% RSLogix 500 project LVD190111.RSS, saved by version 11.00.00.00 %
PROJECT "LINCEBOT"    % processor: MicroLogix 1400 %

PROGRAM FILES
  LAD 2 "MAIN"  43 rungs  % Main Program Routine %
  LAD 4 "PACKAGER"  10 rungs  % normal %
  LAD 6 "TIMING"  11 rungs  % normal %
  LAD 8 "LOOP TIME"  6 rungs
  LAD 10 "AIR PRESUR"  5 rungs
  LAD 12 "ENABLES"  10 rungs
  LAD 14 "SPEED OUT"  12 rungs
  LAD 16 "TOTALCOUNT"  4 rungs
  LAD 18 "TESTTRIG1"  3 rungs
  LAD 20 "TESTTRIG5"  3 rungs
  LAD 22 "TESTTRIG6"  3 rungs
  LAD 24 "NOTUSED"  1 rungs
  LAD 26 "TEST TIME"  11 rungs
  LAD 70 "NOTUSED"  3 rungs  % normal %
  LAD 80 "HSC BOT"  5 rungs
  LAD 90 "HSC TOP"  6 rungs
  LAD 100 "1 MS STI"  27 rungs  % high speed %
  LAD 102 "SPEED BOT"  8 rungs  % high speed %
  LAD 103 "SPEED TOP"  8 rungs  % high speed %
  LAD 104 "P BOT"  9 rungs  % high speed %
  LAD 105 "P TOP"  8 rungs  % high speed %
  LAD 110 "SHIFT BOT"  9 rungs
  LAD 111 "SHIFT TOP"  13 rungs
  LAD 122 "OPTICBOT"  2 rungs
  LAD 124 "INS1RESULT"  6 rungs
  LAD 125 "INS 1 MOVE"  7 rungs
  LAD 126 "INS 1TIME"  36 rungs
  LAD 127 "INS1"  16 rungs
  LAD 128 "INS1PASS"  4 rungs
  LAD 129 "INS1ACQ"  8 rungs
  LAD 130 "INS1TRIG"  5 rungs
  LAD 131 "XFER"  2 rungs
  LAD 141 "OPTICTOP"  13 rungs
  LAD 149 "INS5RESULT"  6 rungs
  LAD 150 "INS 5 MOVE"  11 rungs
  LAD 151 "INS 6 MOVE"  11 rungs
  LAD 152 "INS5"  16 rungs
  LAD 153 "INS5PASS"  4 rungs
  LAD 154 "INS5ACQ"  8 rungs
  LAD 155 "INS5TRIG"  5 rungs
  LAD 159 "INS6RESULT"  6 rungs
  LAD 160 "INS 5 TIME"  42 rungs
  LAD 161 "INS 6 TIME"  42 rungs
  LAD 162 "INS6"  16 rungs
  LAD 163 "INS6PASS"  4 rungs
  LAD 164 "INS6ACQ"  8 rungs
  LAD 165 "INS6TRIG"  5 rungs
  LAD 170 "PASS BLOW"  10 rungs
  LAD 180 "RATE"  9 rungs

DATA FILES
  O0 OUTPUT  11 elements
  I1 INPUT  11 elements
  S2 STATUS  66 elements
  B3 BINARY  14 elements
  T4 TIMER  40 elements
  C5 COUNTER  1 elements
  R6 CONTROL  20 elements
  N7 INTEGER  200 elements
  F8 FLOAT  100 elements
  B9 TOP BS DAT  256 elements
  B10 OLD_COM  1 elements
  B11 BOT BS DAT  256 elements
  B12 HMI_BINARY  22 elements  % general use with hmi to avoid additional reads %
  L13  COUNTS  100 elements
  F14 HMI_FLOATS  100 elements
  N15 HMI_INTS  100 elements
  L16 HMI_LONGS  100 elements
  B17 SIDE DATA  128 elements
  B18 TOP DATA  128 elements
  L19 INS1TIME  10 elements
  L20 INS1POS  10 elements
  L21 INS5TIME  10 elements
  L22 INS5POS  10 elements
  L23 NEW READ  100 elements
  L24 NEW WRITE  100 elements
  L25 INS6TIME  10 elements
  L26 INS6POS  10 elements
  L42   52 elements
  B181 BLANK  128 elements  % used to wipe bs files %
  F182 TEST FLOAT  50 elements
  L183 TEST LONG  50 elements
  N184 TEST INTS  50 elements
  B185 TEST BITS  50 elements
  N186 HMI INTS  50 elements
  L187 HMI LONG  50 elements
  F188 HMI FLOAT  50 elements
  B189 HMI BITS  50 elements
  L190 COUNTS  50 elements
  B191 ERROR BITS  10 elements
  L192 SPD OFFSET  50 elements
  F193 SPD OFFSET  50 elements
  B194 BOT GOOD  128 elements
  B195 TOP GOOD  128 elements
  B196 CTRL BITS  50 elements
  N197 CTRL INTS  50 elements
  B198 TRK BITS  50 elements
  L199 TRK LONG  50 elements
  N200 TRK INTS  50 elements
  L201 INS LONG  50 elements
  B202 INS BITS  50 elements
  N203 INS INTS  50 elements
  L204 CTRL LONG  50 elements
  F205 CTRL FLTS  50 elements

LADDER 2 "MAIN"    % Main Program Routine %
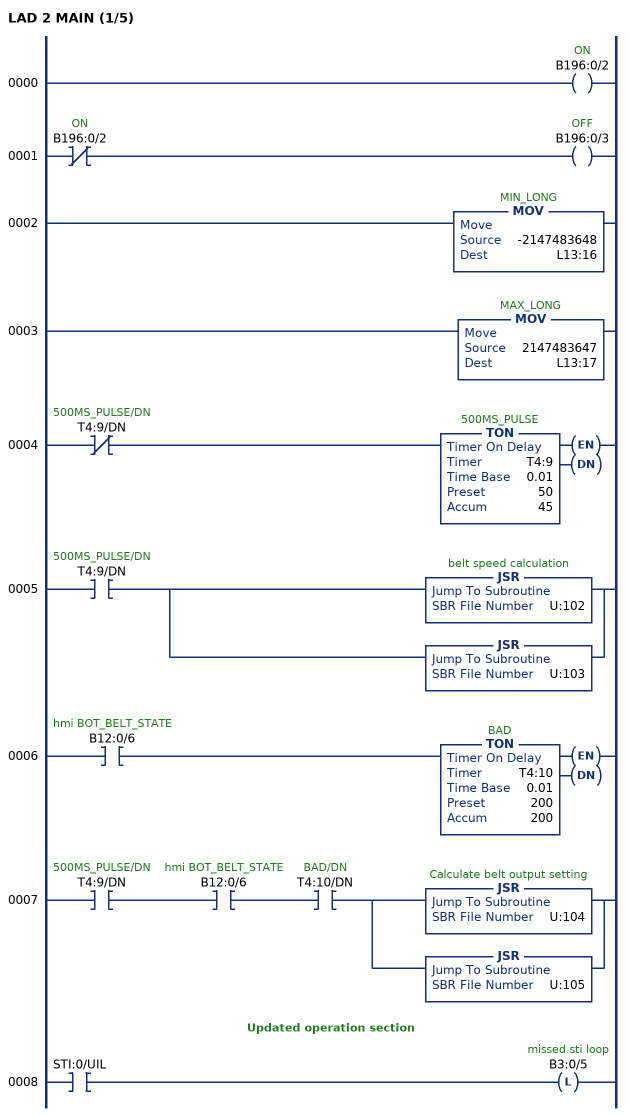
% Rung: 0 %
SOR OTE B196:0/2 EOR
%   B196:0/2  ON %
% Rung: 1 %
SOR XIO B196:0/2 OTE B196:0/3 EOR
%   B196:0/2  ON %
%   B196:0/3  OFF %
% Rung: 2 %
SOR MOV -2147483648 L13:16 EOR
%   L13:16  MIN_LONG %
% Rung: 3 %
SOR MOV 2147483647 L13:17 EOR
%   L13:17  MAX_LONG %
% Rung: 4 %
SOR XIO T4:9/DN TON T4:9 0.01 50 45 EOR
%   T4:9  500MS_PULSE %
% Rung: 5 %
SOR XIC T4:9/DN BST JSR U:102 NXB JSR U:103 BND EOR
%   T4:9  500MS_PULSE %
%   U:102  "belt speed calculation" %
% Rung: 6 %
SOR XIC B12:0/6 TON T4:10 0.01 200 200 EOR
%   B12:0/6  BOT_BELT_STATE  "hmi" %
%   T4:10  BAD %
% Rung: 7 %
SOR XIC T4:9/DN XIC B12:0/6 XIC T4:10/DN BST JSR U:104 NXB JSR U:105 BND EOR
%   T4:9  500MS_PULSE %
%   B12:0/6  BOT_BELT_STATE  "hmi" %
%   T4:10  BAD %
%   U:104  "Calculate belt output setting" %
% Rung: 8 %
% TITLE: Updated operation section %
SOR XIC STI:0/UIL OTL B3:0/5 EOR
%   B3:0/5  "missed sti loop" %

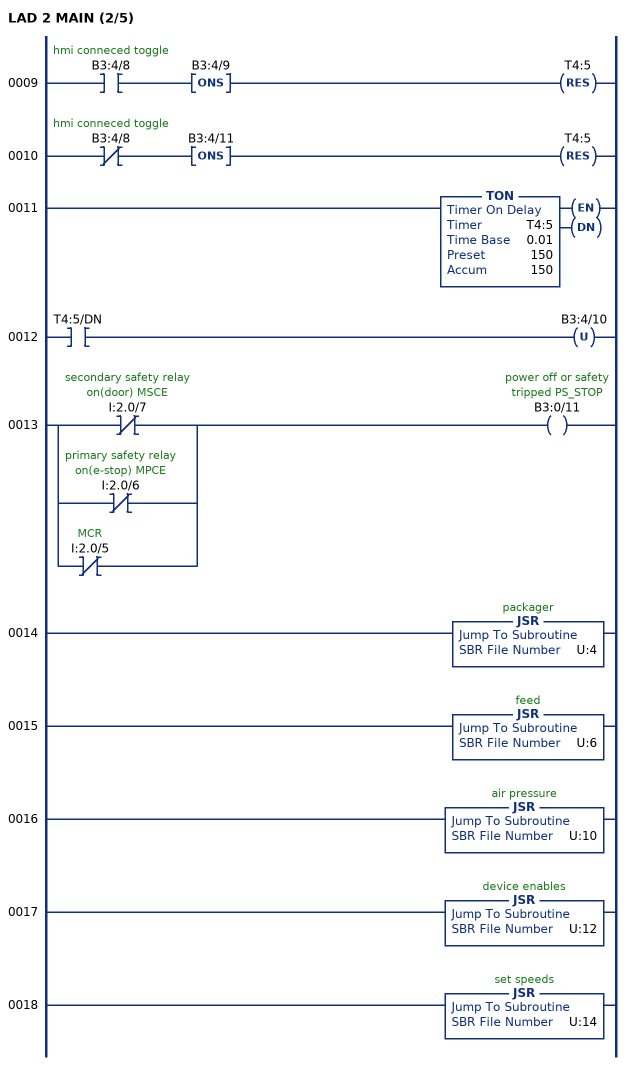
% Rung: 9 %
SOR XIC B3:4/8 ONS B3:4/9 RES T4:5 EOR
%   B3:4/8  "hmi conneced toggle" %
% Rung: 10 %
SOR XIO B3:4/8 ONS B3:4/11 RES T4:5 EOR
%   B3:4/8  "hmi conneced toggle" %
% Rung: 11 %
SOR TON T4:5 0.01 150 150 EOR
% Rung: 12 %
SOR XIC T4:5/DN OTU B3:4/10 EOR
% Rung: 13 %
SOR BST XIO I:2.0/7 NXB XIO I:2.0/6 NXB XIO I:2.0/5 BND OTE B3:0/11 EOR
%   I:2.0/7  MSCE  "secondary safety relay on(door)" %
%   I:2.0/6  MPCE  "primary safety relay on(e-stop)" %
%   I:2.0/5  MCR %
%   B3:0/11  PS_STOP  "power off or safety tripped" %
% Rung: 14 %
SOR JSR U:4 EOR
%   U:4  "packager" %
% Rung: 15 %
SOR JSR U:6 EOR
%   U:6  "feed" %
% Rung: 16 %
SOR JSR U:10 EOR
%   U:10  "air pressure" %
% Rung: 17 %
SOR JSR U:12 EOR
%   U:12  "device enables" %
% Rung: 18 %
SOR JSR U:14 EOR
%   U:14  "set speeds" %

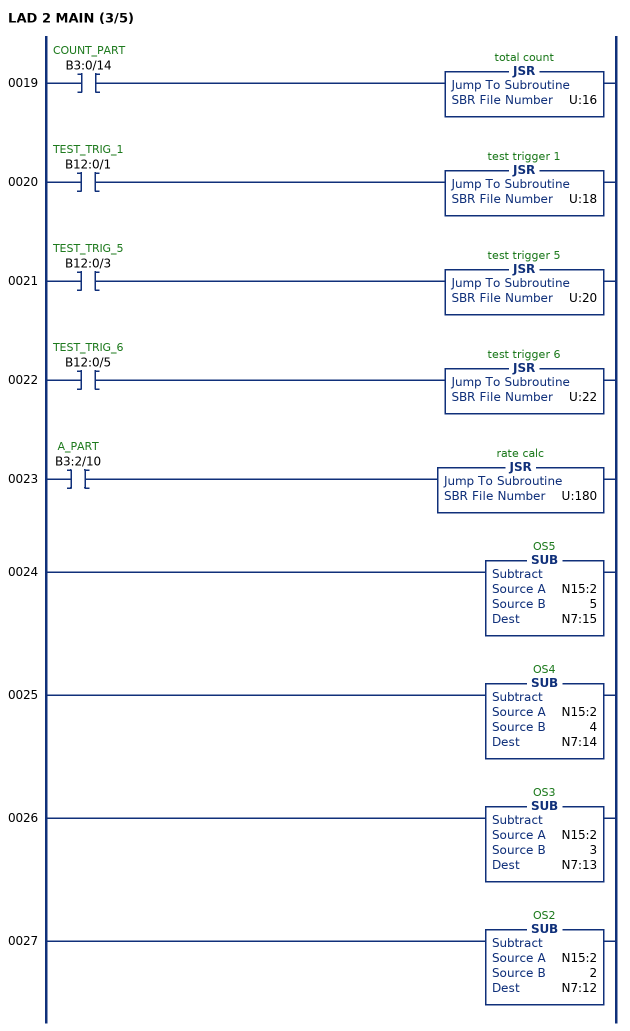
% Rung: 19 %
SOR XIC B3:0/14 JSR U:16 EOR
%   B3:0/14  COUNT_PART %
%   U:16  "total count" %
% Rung: 20 %
SOR XIC B12:0/1 JSR U:18 EOR
%   B12:0/1  TEST_TRIG_1 %
%   U:18  "test trigger 1" %
% Rung: 21 %
SOR XIC B12:0/3 JSR U:20 EOR
%   B12:0/3  TEST_TRIG_5 %
%   U:20  "test trigger 5" %
% Rung: 22 %
SOR XIC B12:0/5 JSR U:22 EOR
%   B12:0/5  TEST_TRIG_6 %
%   U:22  "test trigger 6" %
% Rung: 23 %
SOR XIC B3:2/10 JSR U:180 EOR
%   B3:2/10  A_PART %
%   U:180  "rate calc" %
% Rung: 24 %
SOR SUB N15:2 5 N7:15 EOR
%   N15:2  BLOW_PT %
%   N7:15  OS5 %
% Rung: 25 %
SOR SUB N15:2 4 N7:14 EOR
%   N15:2  BLOW_PT %
%   N7:14  OS4 %
% Rung: 26 %
SOR SUB N15:2 3 N7:13 EOR
%   N15:2  BLOW_PT %
%   N7:13  OS3 %
% Rung: 27 %
SOR SUB N15:2 2 N7:12 EOR
%   N15:2  BLOW_PT %
%   N7:12  OS2 %

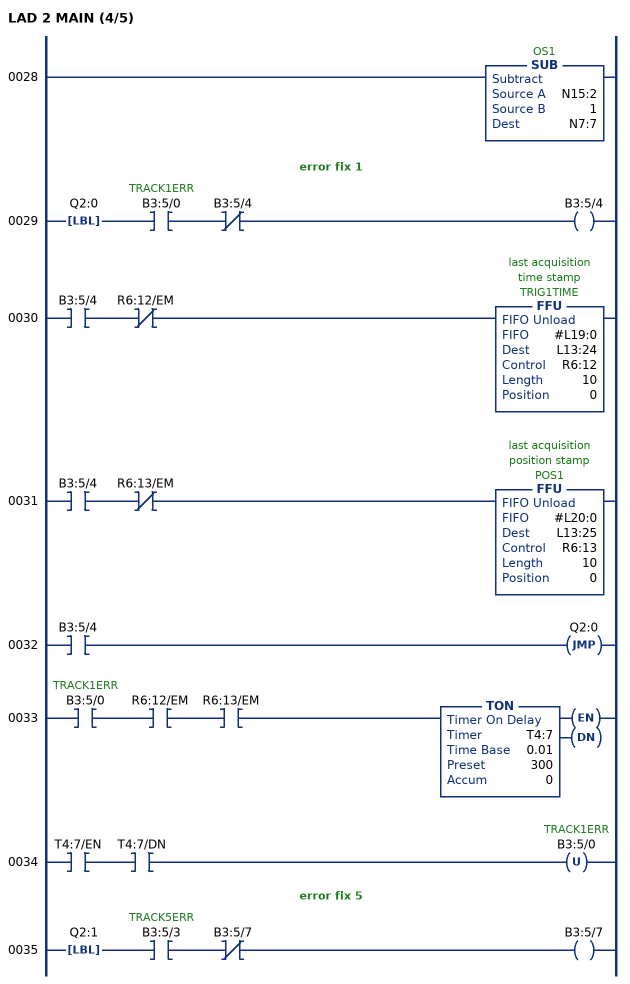
% Rung: 28 %
SOR SUB N15:2 1 N7:7 EOR
%   N15:2  BLOW_PT %
%   N7:7  OS1 %
% Rung: 29 %
% TITLE: error fix 1 %
SOR LBL Q2:0 XIC B3:5/0 XIO B3:5/4 OTE B3:5/4 EOR
%   B3:5/0  TRACK1ERR %
% Rung: 30 %
SOR XIC B3:5/4 XIO R6:12/EM FFU #L19:0 L13:24 R6:12 10 0 EOR
%   L13:24  TRIG1TIME  "last acquisition time stamp" %
% Rung: 31 %
SOR XIC B3:5/4 XIO R6:13/EM FFU #L20:0 L13:25 R6:13 10 0 EOR
%   L13:25  POS1  "last acquisition position stamp" %
% Rung: 32 %
SOR XIC B3:5/4 JMP Q2:0 EOR
% Rung: 33 %
SOR XIC B3:5/0 XIC R6:12/EM XIC R6:13/EM TON T4:7 0.01 300 0 EOR
%   B3:5/0  TRACK1ERR %
% Rung: 34 %
SOR XIC T4:7/EN XIC T4:7/DN OTU B3:5/0 EOR
%   B3:5/0  TRACK1ERR %
% Rung: 35 %
% TITLE: error fix 5 %
SOR LBL Q2:1 XIC B3:5/3 XIO B3:5/7 OTE B3:5/7 EOR
%   B3:5/3  TRACK5ERR %

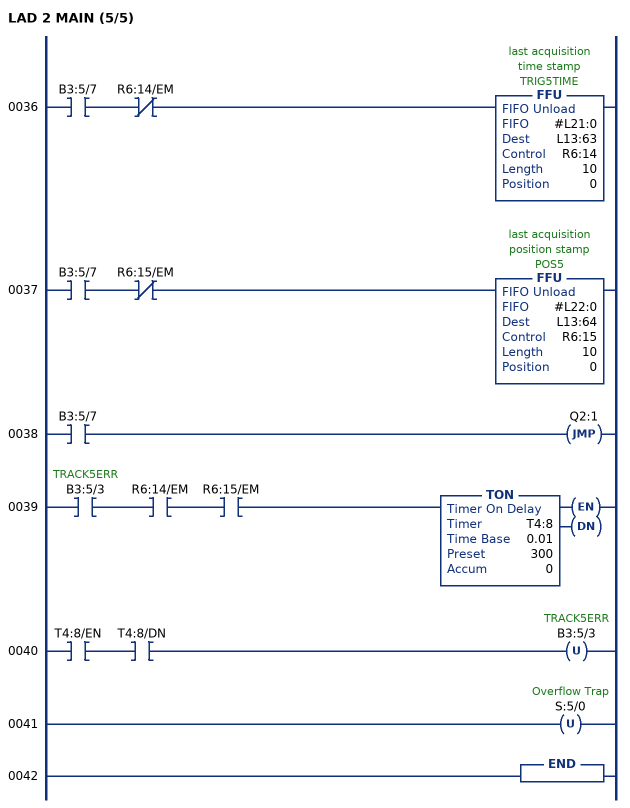
% Rung: 36 %
SOR XIC B3:5/7 XIO R6:14/EM FFU #L21:0 L13:63 R6:14 10 0 EOR
%   L13:63  TRIG5TIME  "last acquisition time stamp" %
% Rung: 37 %
SOR XIC B3:5/7 XIO R6:15/EM FFU #L22:0 L13:64 R6:15 10 0 EOR
%   L13:64  POS5  "last acquisition position stamp" %
% Rung: 38 %
SOR XIC B3:5/7 JMP Q2:1 EOR
% Rung: 39 %
SOR XIC B3:5/3 XIC R6:14/EM XIC R6:15/EM TON T4:8 0.01 300 0 EOR
%   B3:5/3  TRACK5ERR %
% Rung: 40 %
SOR XIC T4:8/EN XIC T4:8/DN OTU B3:5/3 EOR
%   B3:5/3  TRACK5ERR %
% Rung: 41 %
SOR OTU S:5/0 EOR
%   S:5/0  "Overflow Trap" %
% Rung: 42 %
SOR END EOR

LADDER 4 "PACKAGER"    % normal %
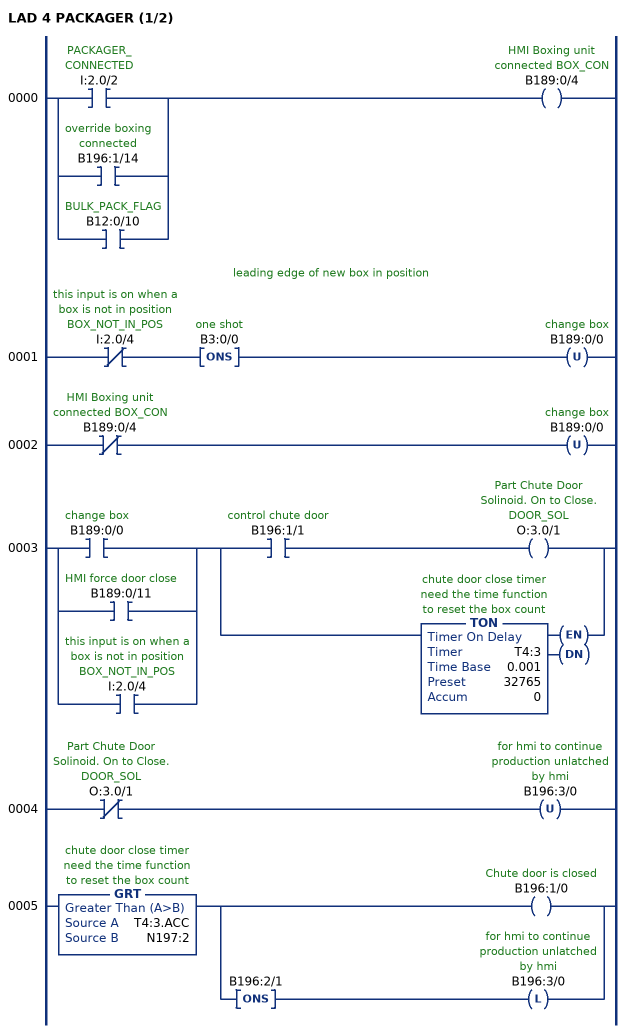
% Rung: 0 %
SOR BST XIC I:2.0/2 NXB XIC B196:1/14 NXB XIC B12:0/10 BND OTE B189:0/4 EOR
%   I:2.0/2  PACKAGER_CONNECTED %
%   B196:1/14  "override boxing connected" %
%   B12:0/10  BULK_PACK_FLAG %
%   B189:0/4  BOX_CON  "HMI Boxing unit connected" %
% Rung: 1 %
% leading edge of new box in position %
SOR XIO I:2.0/4 ONS B3:0/0 OTU B189:0/0 EOR
%   I:2.0/4  BOX_NOT_IN_POS  "this input is on when a box is not in position" %
%   B3:0/0  "one shot" %
%   B189:0/0  "change box" %
% Rung: 2 %
SOR XIO B189:0/4 OTU B189:0/0 EOR
%   B189:0/4  BOX_CON  "HMI Boxing unit connected" %
%   B189:0/0  "change box" %
% Rung: 3 %
SOR BST XIC B189:0/0 NXB XIC B189:0/11 NXB XIC I:2.0/4 BND BST XIC B196:1/1 OTE O:3.0/1 NXB TON T4:3 0.001 32765 0 BND EOR
%   B189:0/0  "change box" %
%   B189:0/11  "HMI force door close" %
%   I:2.0/4  BOX_NOT_IN_POS  "this input is on when a box is not in position" %
%   B196:1/1  "control chute door" %
%   O:3.0/1  DOOR_SOL  "Part Chute Door Solinoid. On to Close." %
%   T4:3  "chute door close timer need the time function to reset the box count" %
% Rung: 4 %
SOR XIO O:3.0/1 OTU B196:3/0 EOR
%   O:3.0/1  DOOR_SOL  "Part Chute Door Solinoid. On to Close." %
%   B196:3/0  "for hmi to continue production unlatched by hmi" %
% Rung: 5 %
SOR GRT T4:3.ACC N197:2 BST OTE B196:1/0 NXB ONS B196:2/1 OTL B196:3/0 BND EOR
%   T4:3  "chute door close timer need the time function to reset the box count" %
%   N197:2  "time for chute door to close" %
%   B196:1/0  "Chute door is closed" %
%   B196:3/0  "for hmi to continue production unlatched by hmi" %

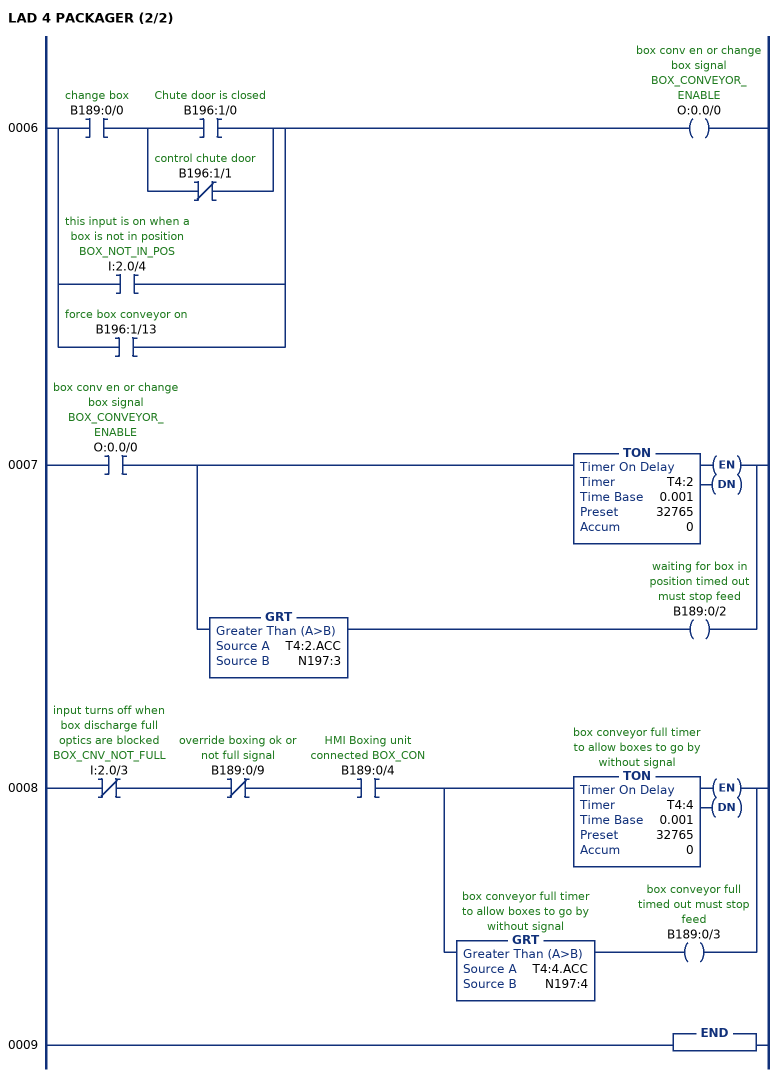
% Rung: 6 %
SOR BST XIC B189:0/0 BST XIC B196:1/0 NXB XIO B196:1/1 BND NXB XIC I:2.0/4 NXB XIC B196:1/13 BND OTE O:0.0/0 EOR
%   B189:0/0  "change box" %
%   B196:1/0  "Chute door is closed" %
%   B196:1/1  "control chute door" %
%   I:2.0/4  BOX_NOT_IN_POS  "this input is on when a box is not in position" %
%   B196:1/13  "force box conveyor on" %
%   O:0.0/0  BOX_CONVEYOR_ENABLE  "box conv en or change box signal" %
% Rung: 7 %
SOR XIC O:0.0/0 BST TON T4:2 0.001 32765 0 NXB GRT T4:2.ACC N197:3 OTE B189:0/2 BND EOR
%   O:0.0/0  BOX_CONVEYOR_ENABLE  "box conv en or change box signal" %
%   N197:3  "FeedWheel Speed Output Setting" %
%   B189:0/2  "waiting for box in position timed out must stop feed" %
% Rung: 8 %
SOR XIO I:2.0/3 XIO B189:0/9 XIC B189:0/4 BST TON T4:4 0.001 32765 0 NXB GRT T4:4.ACC N197:4 OTE B189:0/3 BND EOR
%   I:2.0/3  BOX_CNV_NOT_FULL  "input turns off when box discharge full optics are blocked" %
%   B189:0/9  "override boxing ok or not full signal" %
%   B189:0/4  BOX_CON  "HMI Boxing unit connected" %
%   T4:4  "box conveyor full timer to allow boxes to go by without signal" %
%   N197:4  "boxing convery full time out time (ms)" %
%   B189:0/3  "box conveyor full timed out must stop feed" %
% Rung: 9 %
SOR END EOR

LADDER 6 "TIMING"    % normal %
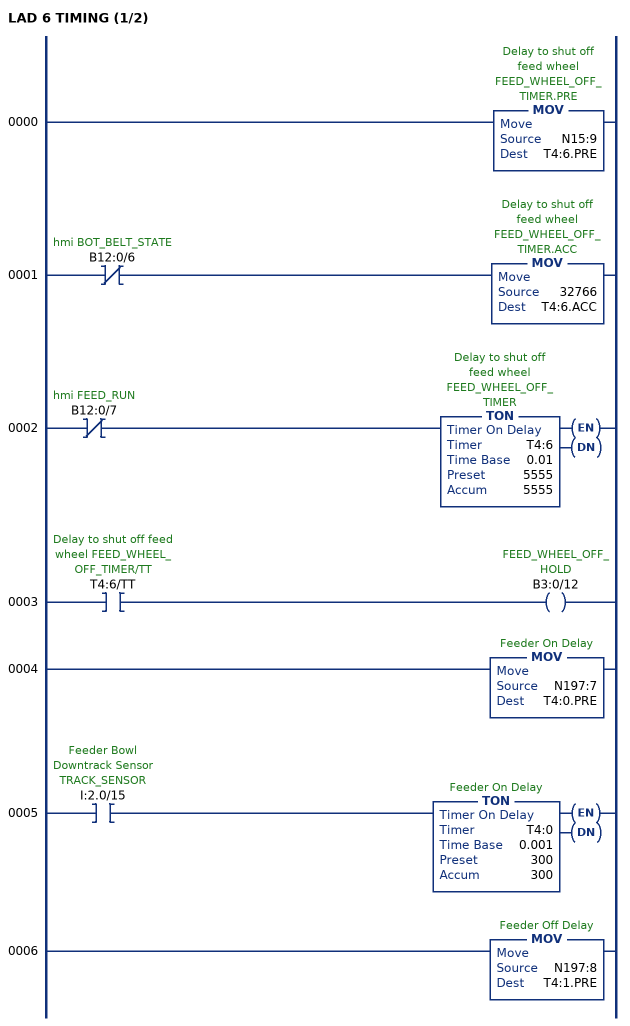
% Rung: 0 %
SOR MOV N15:9 T4:6.PRE EOR
%   N15:9  FEED_WHEEL_STOP_TIME %
%   T4:6  FEED_WHEEL_OFF_TIMER  "Delay to shut off feed wheel" %
% Rung: 1 %
SOR XIO B12:0/6 MOV 32766 T4:6.ACC EOR
%   B12:0/6  BOT_BELT_STATE  "hmi" %
%   T4:6  FEED_WHEEL_OFF_TIMER  "Delay to shut off feed wheel" %
% Rung: 2 %
SOR XIO B12:0/7 TON T4:6 0.01 5555 5555 EOR
%   B12:0/7  FEED_RUN  "hmi" %
%   T4:6  FEED_WHEEL_OFF_TIMER  "Delay to shut off feed wheel" %
% Rung: 3 %
SOR XIC T4:6/TT OTE B3:0/12 EOR
%   T4:6  FEED_WHEEL_OFF_TIMER  "Delay to shut off feed wheel" %
%   B3:0/12  FEED_WHEEL_OFF_HOLD %
% Rung: 4 %
SOR MOV N197:7 T4:0.PRE EOR
%   N197:7  "down track on delay" %
%   T4:0  "Feeder On Delay" %
% Rung: 5 %
SOR XIC I:2.0/15 TON T4:0 0.001 300 300 EOR
%   I:2.0/15  TRACK_SENSOR  "Feeder Bowl Downtrack Sensor" %
%   T4:0  "Feeder On Delay" %
% Rung: 6 %
SOR MOV N197:8 T4:1.PRE EOR
%   N197:8  "down track off delay" %
%   T4:1  "Feeder Off Delay" %

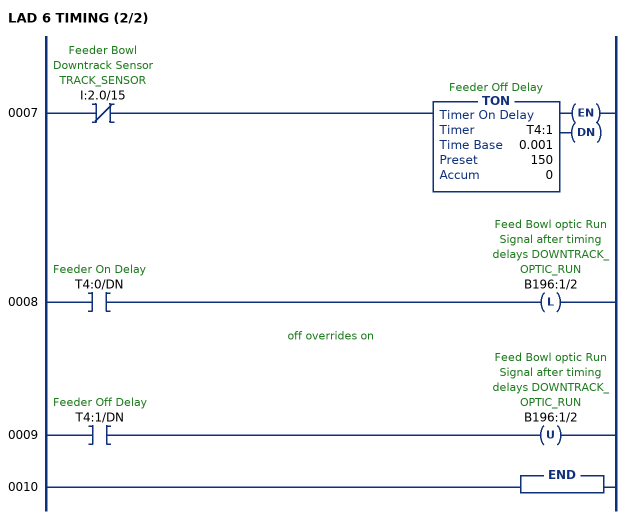
% Rung: 7 %
SOR XIO I:2.0/15 TON T4:1 0.001 150 0 EOR
%   I:2.0/15  TRACK_SENSOR  "Feeder Bowl Downtrack Sensor" %
%   T4:1  "Feeder Off Delay" %
% Rung: 8 %
SOR XIC T4:0/DN OTL B196:1/2 EOR
%   T4:0  "Feeder On Delay" %
%   B196:1/2  DOWNTRACK_OPTIC_RUN  "Feed Bowl optic Run Signal after timing delays" %
% Rung: 9 %
% off overrides on %
SOR XIC T4:1/DN OTU B196:1/2 EOR
%   T4:1  "Feeder Off Delay" %
%   B196:1/2  DOWNTRACK_OPTIC_RUN  "Feed Bowl optic Run Signal after timing delays" %
% Rung: 10 %
SOR END EOR

LADDER 8 "LOOP TIME"
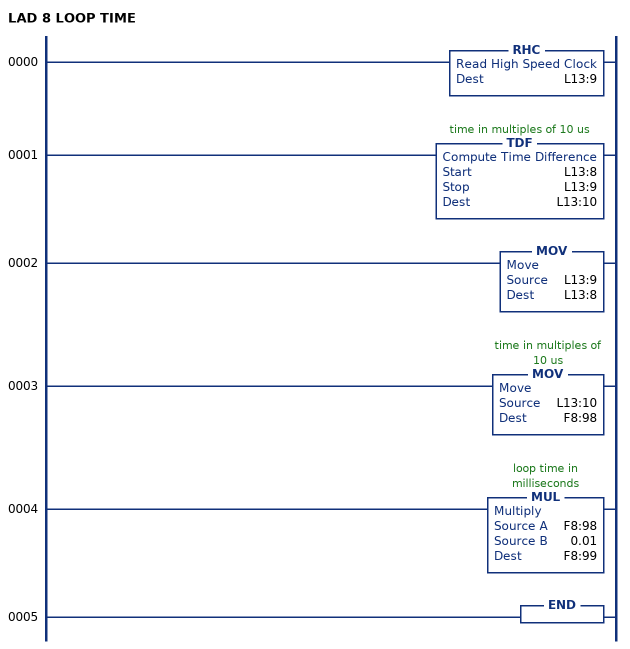
% Rung: 0 %
SOR RHC L13:9 EOR
% Rung: 1 %
SOR TDF L13:8 L13:9 L13:10 EOR
%   L13:10  "time in multiples of 10 us" %
% Rung: 2 %
SOR MOV L13:9 L13:8 EOR
% Rung: 3 %
SOR MOV L13:10 F8:98 EOR
%   L13:10  "time in multiples of 10 us" %
%   F8:98  "time in multiples of 10 us" %
% Rung: 4 %
SOR MUL F8:98 0.01 F8:99 EOR
%   F8:98  "time in multiples of 10 us" %
%   F8:99  "loop time in milliseconds" %
% Rung: 5 %
SOR END EOR

LADDER 10 "AIR PRESUR"
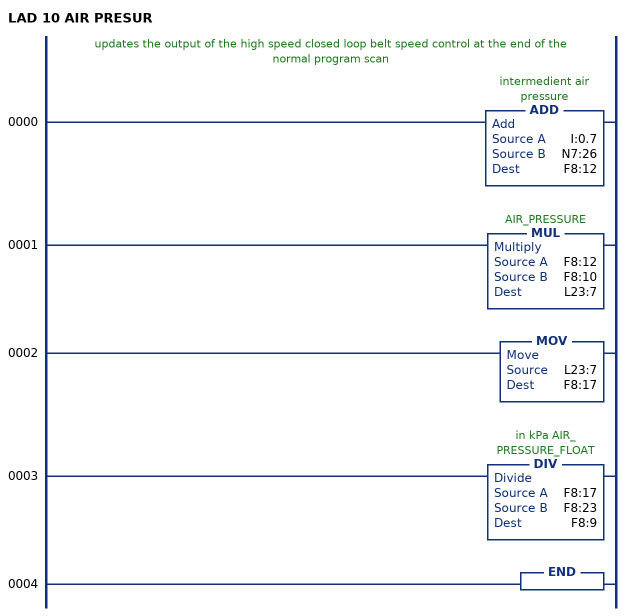
% Rung: 0 %
% updates the output of the high speed closed loop belt speed control at the end of the normal program scan %
SOR ADD I:0.7 N7:26 F8:12 EOR
%   I:0.7  "Air Presure Sensor Input Signal" %
%   N7:26  MAIN_AIR_OFFSET  "Main Air Offset old machine -398 new machine 0" %
%   F8:12  "intermedient air pressure" %
% Rung: 1 %
SOR MUL F8:12 F8:10 L23:7 EOR
%   F8:12  "intermedient air pressure" %
%   F8:10  AIR_MULTIPLIER_BAR  "Air Multiplier (BAR)" %
%   L23:7  AIR_PRESSURE %
% Rung: 2 %
SOR MOV L23:7 F8:17 EOR
%   L23:7  AIR_PRESSURE %
% Rung: 3 %
SOR DIV F8:17 F8:23 F8:9 EOR
%   F8:9  AIR_PRESSURE_FLOAT  "in kPa" %
% Rung: 4 %
SOR END EOR

LADDER 12 "ENABLES"
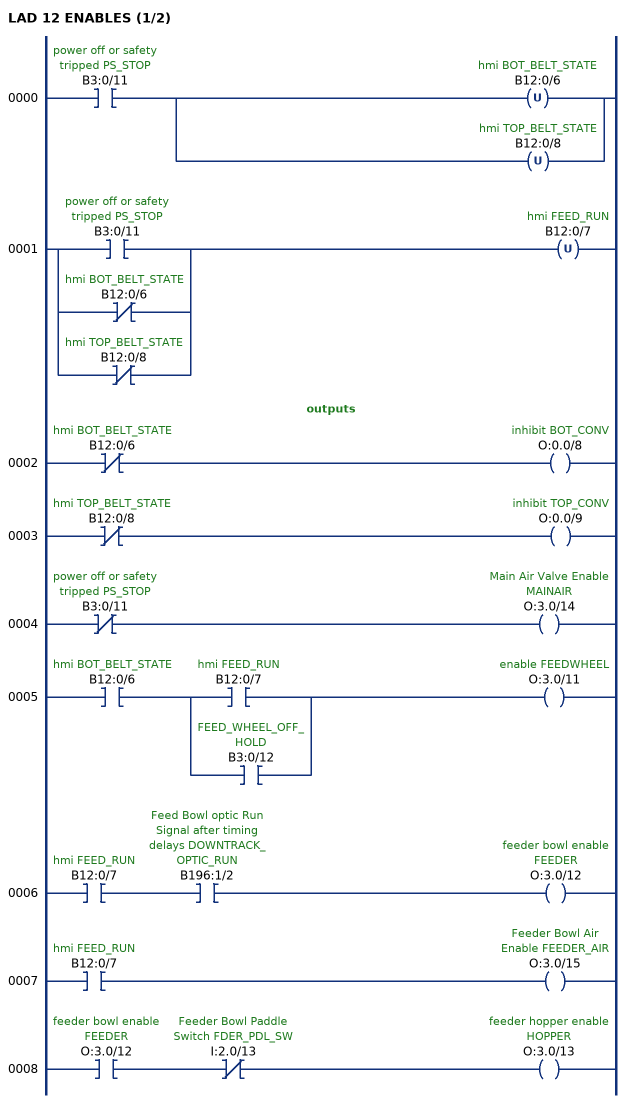
% Rung: 0 %
SOR XIC B3:0/11 BST OTU B12:0/6 NXB OTU B12:0/8 BND EOR
%   B3:0/11  PS_STOP  "power off or safety tripped" %
%   B12:0/6  BOT_BELT_STATE  "hmi" %
%   B12:0/8  TOP_BELT_STATE  "hmi" %
% Rung: 1 %
SOR BST XIC B3:0/11 NXB XIO B12:0/6 NXB XIO B12:0/8 BND OTU B12:0/7 EOR
%   B3:0/11  PS_STOP  "power off or safety tripped" %
%   B12:0/6  BOT_BELT_STATE  "hmi" %
%   B12:0/8  TOP_BELT_STATE  "hmi" %
%   B12:0/7  FEED_RUN  "hmi" %
% Rung: 2 %
% TITLE: outputs %
SOR XIO B12:0/6 OTE O:0.0/8 EOR
%   B12:0/6  BOT_BELT_STATE  "hmi" %
%   O:0.0/8  BOT_CONV  "inhibit" %
% Rung: 3 %
SOR XIO B12:0/8 OTE O:0.0/9 EOR
%   B12:0/8  TOP_BELT_STATE  "hmi" %
%   O:0.0/9  TOP_CONV  "inhibit" %
% Rung: 4 %
SOR XIO B3:0/11 OTE O:3.0/14 EOR
%   B3:0/11  PS_STOP  "power off or safety tripped" %
%   O:3.0/14  MAINAIR  "Main Air Valve Enable" %
% Rung: 5 %
SOR XIC B12:0/6 BST XIC B12:0/7 NXB XIC B3:0/12 BND OTE O:3.0/11 EOR
%   B12:0/6  BOT_BELT_STATE  "hmi" %
%   B12:0/7  FEED_RUN  "hmi" %
%   B3:0/12  FEED_WHEEL_OFF_HOLD %
%   O:3.0/11  FEEDWHEEL  "enable" %
% Rung: 6 %
SOR XIC B12:0/7 XIC B196:1/2 OTE O:3.0/12 EOR
%   B12:0/7  FEED_RUN  "hmi" %
%   B196:1/2  DOWNTRACK_OPTIC_RUN  "Feed Bowl optic Run Signal after timing delays" %
%   O:3.0/12  FEEDER  "feeder bowl enable" %
% Rung: 7 %
SOR XIC B12:0/7 OTE O:3.0/15 EOR
%   B12:0/7  FEED_RUN  "hmi" %
%   O:3.0/15  FEEDER_AIR  "Feeder Bowl Air Enable" %
% Rung: 8 %
SOR XIC O:3.0/12 XIO I:2.0/13 OTE O:3.0/13 EOR
%   O:3.0/12  FEEDER  "feeder bowl enable" %
%   I:2.0/13  FDER_PDL_SW  "Feeder Bowl Paddle Switch" %
%   O:3.0/13  HOPPER  "feeder hopper enable" %

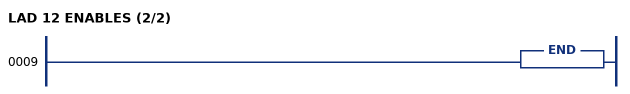
% Rung: 9 %
SOR END EOR

LADDER 14 "SPEED OUT"
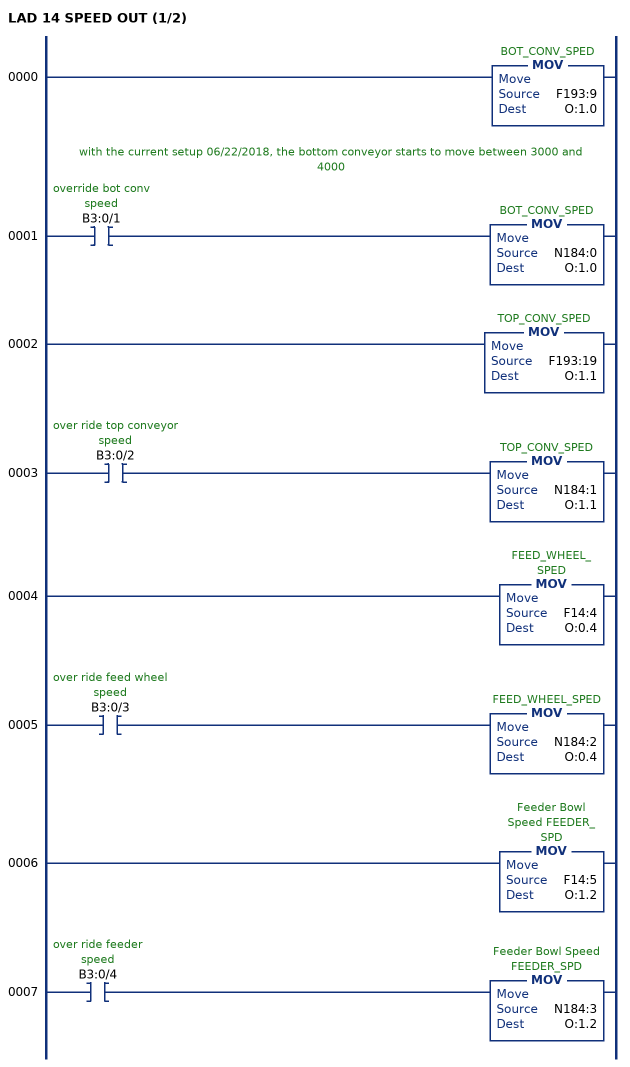
% Rung: 0 %
SOR MOV F193:9 O:1.0 EOR
%   F193:9  SCALED_BOT_VALUE %
%   O:1.0  BOT_CONV_SPED %
% Rung: 1 %
% with the current setup 06/22/2018, the bottom conveyor starts to move between 3000 and 4000 %
SOR XIC B3:0/1 MOV N184:0 O:1.0 EOR
%   B3:0/1  "override bot conv speed" %
%   O:1.0  BOT_CONV_SPED %
% Rung: 2 %
SOR MOV F193:19 O:1.1 EOR
%   F193:19  SCALED_TOP_VALUE %
%   O:1.1  TOP_CONV_SPED %
% Rung: 3 %
SOR XIC B3:0/2 MOV N184:1 O:1.1 EOR
%   B3:0/2  "over ride top conveyor speed" %
%   O:1.1  TOP_CONV_SPED %
% Rung: 4 %
SOR MOV F14:4 O:0.4 EOR
%   O:0.4  FEED_WHEEL_SPED %
% Rung: 5 %
SOR XIC B3:0/3 MOV N184:2 O:0.4 EOR
%   B3:0/3  "over ride feed wheel speed" %
%   O:0.4  FEED_WHEEL_SPED %
% Rung: 6 %
SOR MOV F14:5 O:1.2 EOR
%   O:1.2  FEEDER_SPD  "Feeder Bowl Speed" %
% Rung: 7 %
SOR XIC B3:0/4 MOV N184:3 O:1.2 EOR
%   B3:0/4  "over ride feeder speed" %
%   O:1.2  FEEDER_SPD  "Feeder Bowl Speed" %

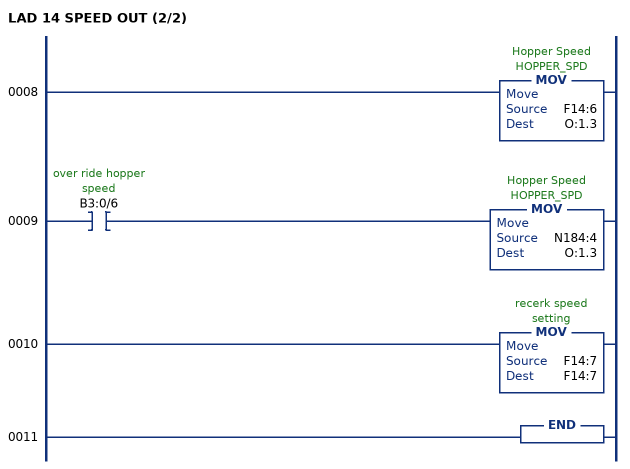
% Rung: 8 %
SOR MOV F14:6 O:1.3 EOR
%   O:1.3  HOPPER_SPD  "Hopper Speed" %
% Rung: 9 %
SOR XIC B3:0/6 MOV N184:4 O:1.3 EOR
%   B3:0/6  "over ride hopper speed" %
%   O:1.3  HOPPER_SPD  "Hopper Speed" %
% Rung: 10 %
SOR MOV F14:7 F14:7 EOR
%   F14:7  "recerk speed setting" %
% Rung: 11 %
SOR END EOR

LADDER 16 "TOTALCOUNT"
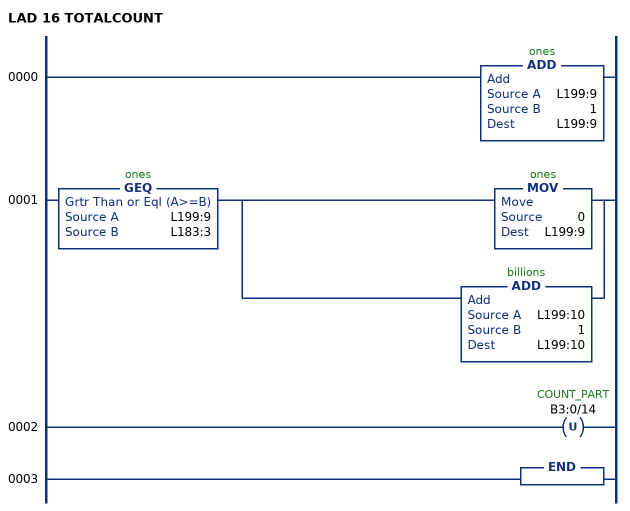
% Rung: 0 %
SOR ADD L199:9 1 L199:9 EOR
%   L199:9  "ones" %
% Rung: 1 %
SOR GEQ L199:9 L183:3 BST MOV 0 L199:9 NXB ADD L199:10 1 L199:10 BND EOR
%   L199:9  "ones" %
%   L183:3  "button state" %
%   L199:10  "billions" %
% Rung: 2 %
SOR OTU B3:0/14 EOR
%   B3:0/14  COUNT_PART %
% Rung: 3 %
SOR END EOR

LADDER 18 "TESTTRIG1"
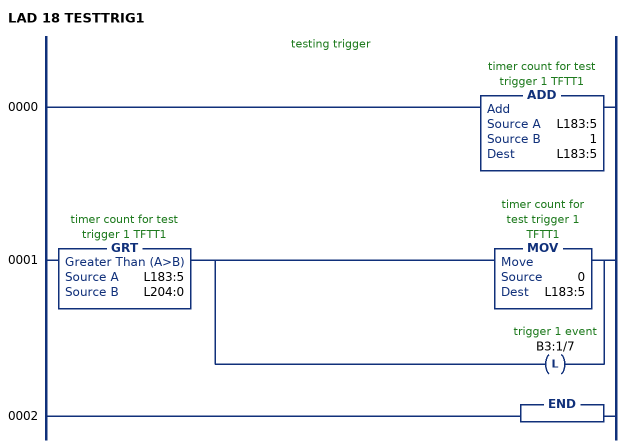
% Rung: 0 %
% testing trigger %
SOR ADD L183:5 1 L183:5 EOR
%   L183:5  TFTT1  "timer count for test trigger 1" %
% Rung: 1 %
SOR GRT L183:5 L204:0 BST MOV 0 L183:5 NXB OTL B3:1/7 BND EOR
%   L183:5  TFTT1  "timer count for test trigger 1" %
%   B3:1/7  "trigger 1 event" %
% Rung: 2 %
SOR END EOR

LADDER 20 "TESTTRIG5"
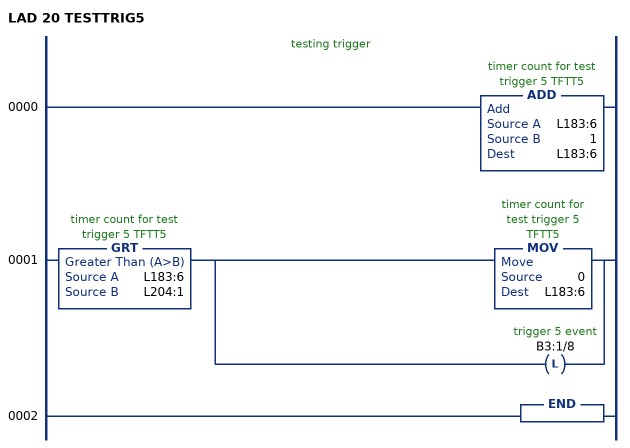
% Rung: 0 %
% testing trigger %
SOR ADD L183:6 1 L183:6 EOR
%   L183:6  TFTT5  "timer count for test trigger 5" %
% Rung: 1 %
SOR GRT L183:6 L204:1 BST MOV 0 L183:6 NXB OTL B3:1/8 BND EOR
%   L183:6  TFTT5  "timer count for test trigger 5" %
%   L204:1  TTT5 %
%   B3:1/8  "trigger 5 event" %
% Rung: 2 %
SOR END EOR

LADDER 22 "TESTTRIG6"
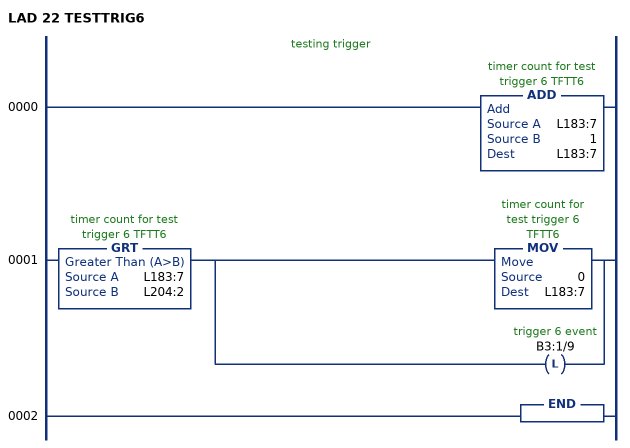
% Rung: 0 %
% testing trigger %
SOR ADD L183:7 1 L183:7 EOR
%   L183:7  TFTT6  "timer count for test trigger 6" %
% Rung: 1 %
SOR GRT L183:7 L204:2 BST MOV 0 L183:7 NXB OTL B3:1/9 BND EOR
%   L183:7  TFTT6  "timer count for test trigger 6" %
%   L204:2  TTT6 %
%   B3:1/9  "trigger 6 event" %
% Rung: 2 %
SOR END EOR

LADDER 26 "TEST TIME"
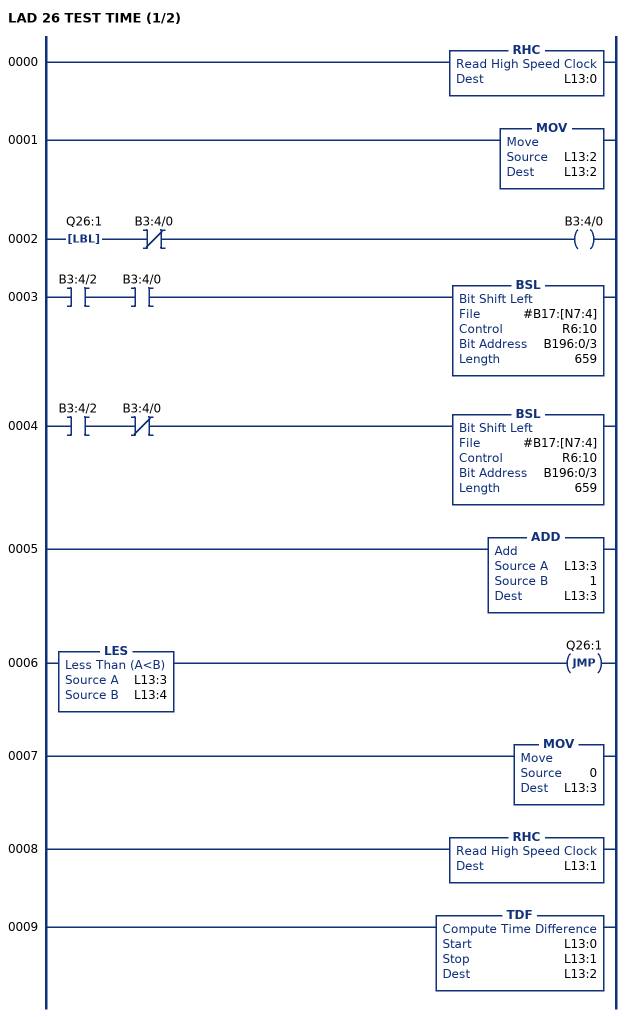
% Rung: 0 %
SOR RHC L13:0 EOR
% Rung: 1 %
SOR MOV L13:2 L13:2 EOR
% Rung: 2 %
SOR LBL Q26:1 XIO B3:4/0 OTE B3:4/0 EOR
% Rung: 3 %
SOR XIC B3:4/2 XIC B3:4/0 BSL #B17:[N7:4] R6:10 B196:0/3 659 EOR
%   B196:0/3  OFF %
% Rung: 4 %
SOR XIC B3:4/2 XIO B3:4/0 BSL #B17:[N7:4] R6:10 B196:0/3 659 EOR
%   B196:0/3  OFF %
% Rung: 5 %
SOR ADD L13:3 1 L13:3 EOR
% Rung: 6 %
SOR LES L13:3 L13:4 JMP Q26:1 EOR
% Rung: 7 %
SOR MOV 0 L13:3 EOR
% Rung: 8 %
SOR RHC L13:1 EOR
% Rung: 9 %
SOR TDF L13:0 L13:1 L13:2 EOR

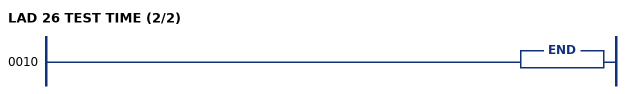
% Rung: 10 %
SOR END EOR

LADDER 70 "NOTUSED"    % normal %
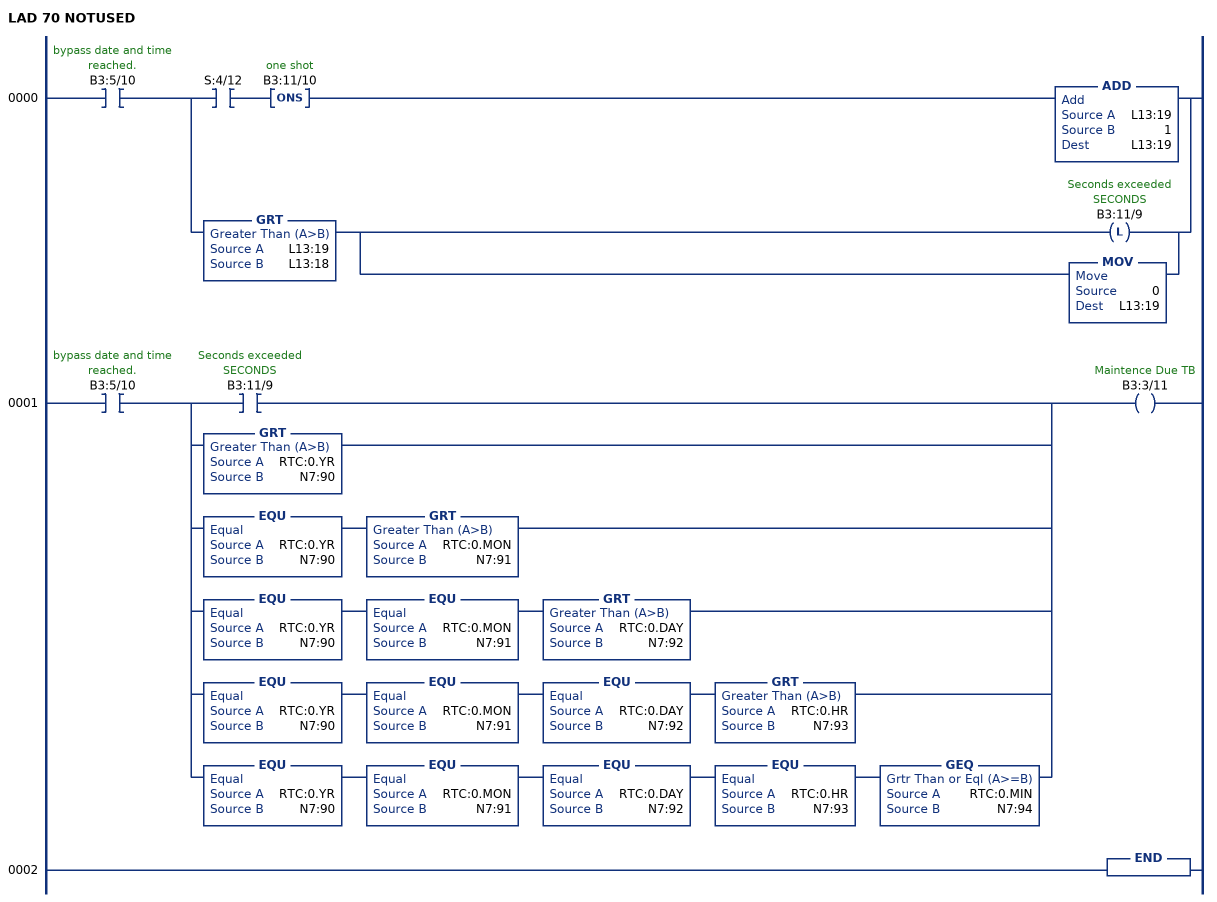
% Rung: 0 %
SOR XIC B3:5/10 BST XIC S:4/12 ONS B3:11/10 ADD L13:19 1 L13:19 NXB GRT L13:19 L13:18 BST OTL B3:11/9 NXB MOV 0 L13:19 BND BND EOR
%   B3:5/10  "bypass date and time reached." %
%   B3:11/10  "one shot" %
%   L13:18  MAX %
%   B3:11/9  SECONDS  "Seconds exceeded" %
% Rung: 1 %
SOR XIC B3:5/10 BST XIC B3:11/9 NXB GRT RTC:0.YR N7:90 NXB EQU RTC:0.YR N7:90 GRT RTC:0.MON N7:91 NXB EQU RTC:0.YR N7:90 EQU RTC:0.MON N7:91 GRT RTC:0.DAY N7:92 NXB EQU RTC:0.YR N7:90 EQU RTC:0.MON N7:91 EQU RTC:0.DAY N7:92 GRT RTC:0.HR N7:93 NXB EQU RTC:0.YR N7:90 EQU RTC:0.MON N7:91 EQU RTC:0.DAY N7:92 EQU RTC:0.HR N7:93 GEQ RTC:0.MIN N7:94 BND OTE B3:3/11 EOR
%   B3:5/10  "bypass date and time reached." %
%   B3:11/9  SECONDS  "Seconds exceeded" %
%   N7:90  RTC %
%   B3:3/11  TB  "Maintence Due" %
% Rung: 2 %
SOR END EOR

LADDER 80 "HSC BOT"
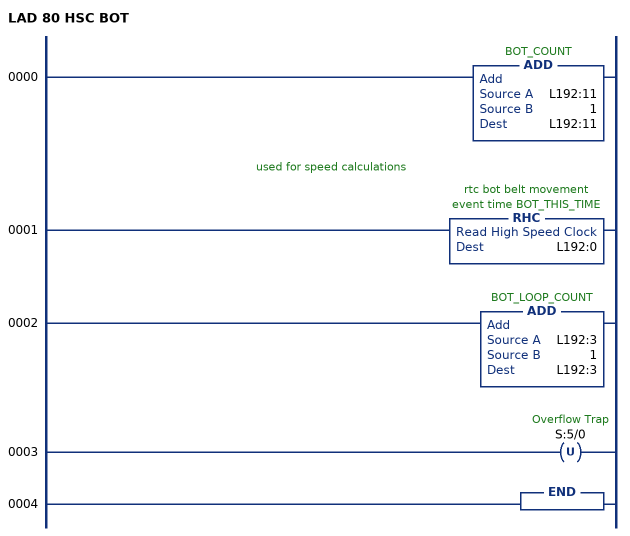
% Rung: 0 %
SOR ADD L192:11 1 L192:11 EOR
%   L192:11  BOT_COUNT %
% Rung: 1 %
% used for speed calculations %
SOR RHC L192:0 EOR
%   L192:0  BOT_THIS_TIME  "rtc bot belt movement event time" %
% Rung: 2 %
SOR ADD L192:3 1 L192:3 EOR
%   L192:3  BOT_LOOP_COUNT %
% Rung: 3 %
SOR OTU S:5/0 EOR
%   S:5/0  "Overflow Trap" %
% Rung: 4 %
SOR END EOR

LADDER 90 "HSC TOP"
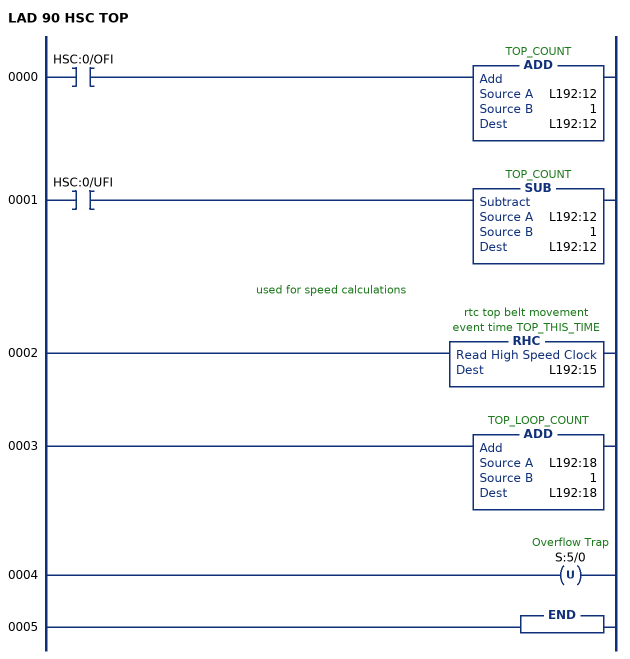
% Rung: 0 %
SOR XIC HSC:0/OFI ADD L192:12 1 L192:12 EOR
%   L192:12  TOP_COUNT %
% Rung: 1 %
SOR XIC HSC:0/UFI SUB L192:12 1 L192:12 EOR
%   L192:12  TOP_COUNT %
% Rung: 2 %
% used for speed calculations %
SOR RHC L192:15 EOR
%   L192:15  TOP_THIS_TIME  "rtc top belt movement event time" %
% Rung: 3 %
SOR ADD L192:18 1 L192:18 EOR
%   L192:18  TOP_LOOP_COUNT %
% Rung: 4 %
SOR OTU S:5/0 EOR
%   S:5/0  "Overflow Trap" %
% Rung: 5 %
SOR END EOR

LADDER 100 "1 MS STI"    % high speed %
